// Interface that defines the standard structure for indexable collections
INTERFACE I_Iterable EXTENDS __SYSTEM.IQueryInterface

// Index of the first element.
PROPERTY _Begin : T_Position
GET
END_GET
END_PROPERTY

// Index of the last element.
PROPERTY _End : T_Position
GET
END_GET
END_PROPERTY

END_INTERFACE

(* stored: Version 1.1.0.1
   Itf I_Iterable: Id {1bb73574-f693-03e6-321d-522590609df2}
   Property _Begin: Id {73321905-0f2e-0407-00aa-91048e6eff82}
   Get Get: Id {8d8c254e-4b6e-0859-2854-cb761631fcfe}
   Property _End: Id {fd9a7466-3c98-02f5-23f1-a7caf2aecf29}
   Get Get: Id {0fcaa15c-f86d-066b-2610-50d35d581457} *)
